{attribute addProperty BoxType "EJ3255-0000-0023"}
{attribute addProperty Id "AI_Standard_ChannelAT %I*ARRAY[0..8] OF AI_Standard_Channel_087F71C7160200WcStateAT %I*WcState_98A4DF7520.250InfoDataAT %I*InfoData_BC63D37F80100"}
{attribute addProperty CRC "220768616"}
{attribute addProperty SizeInBites "242"}
{attribute addProperty SizeInBytes "30.25"}
TYPE EJ3255_7B3AD958 :
STRUCT
	{attribute addProperty Name "AI_Standard_Channel"}
	AI_Standard_Channel : ARRAY[0..8] OF AI_Standard_Channel_087F71C7;
	{attribute addProperty Name "WcState"}
	WcState : WcState_98A4DF75;
	{attribute addProperty Name "InfoData"}
	InfoData : InfoData_BC63D37F;
END_STRUCT
END_TYPE

(* stored: Version 1.2.0.0, ProductVersion 3.1.4024.9
   DUT EJ3255_7B3AD958: Id {6c25dad7-fad8-458a-ac05-74e1f33925e9} *)
